// TIA Portal project "PLC Switching Logic" (V17)
// Pushbuttons Control Outputs? PLC Switching Logic

(* hardware
DEVICE "S7-1200 station_1"  S7-1200 Station
   slot 0: "Rack_0"  S7-1200 Rack  Rack  V1.0
   slot 1: "PLC_1"  CPU 1212C DC/DC/DC  6ES7 212-1AE40-0XB0  V4.5
*)

// ===== PLC "PLC_1"  CPU 1212C DC/DC/DC =====

VAR_GLOBAL   // PLC tag table "Default tag table"
   "Switch PB" AT %I0.0 : Bool;
   "Light" AT %Q0.0 : Bool;
   "Tag_1" AT %M0.0 : Bool;
   "Tag_2" AT %M0.1 : Bool;
   "Tag_3" AT %M0.2 : Bool;
   "Tag_4" AT %M0.3 : Bool;
END_VAR

ORGANIZATION_BLOCK "Main"   // OB1, LAD, ProgramCycle
TITLE = "Main Program Sweep (Cycle)"
{ S7_Optimized_Access := 'TRUE' }
VERSION : 0.1
   VAR_INPUT
      Initial_Call : Bool;   // Initial call of this OB
      Remanence : Bool;   // =True, if remanent data are available
   END_VAR
BEGIN

REGION Network 1
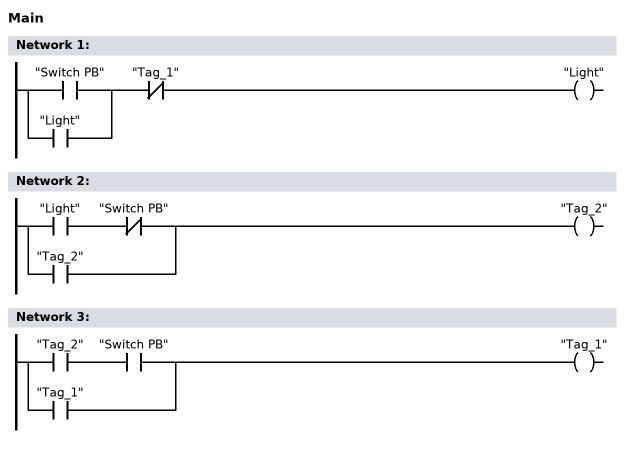
   RUNG wire#powerrail
      Contact( "Switch PB" )
      wire#w1
      I_Contact( "Tag_1" )
      Coil( "Light" )
   END_RUNG
   RUNG wire#powerrail
      Contact( "Light" )
   END_RUNG wire#w1
   // the same network as SCL:
   "Light" := ("Switch PB" OR "Light") AND NOT "Tag_1";
END_REGION

REGION Network 2
   RUNG wire#powerrail
      Contact( "Light" )
      I_Contact( "Switch PB" )
      wire#w1
      Coil( "Tag_2" )
   END_RUNG
   RUNG wire#powerrail
      Contact( "Tag_2" )
   END_RUNG wire#w1
   // the same network as SCL:
   "Tag_2" := ("Light" AND NOT "Switch PB") OR "Tag_2";
END_REGION

REGION Network 3
   RUNG wire#powerrail
      Contact( "Tag_2" )
      Contact( "Switch PB" )
      wire#w1
      Coil( "Tag_1" )
   END_RUNG
   RUNG wire#powerrail
      Contact( "Tag_1" )
   END_RUNG wire#w1
   // the same network as SCL:
   "Tag_1" := ("Tag_2" AND "Switch PB") OR "Tag_1";
END_REGION
END_ORGANIZATION_BLOCK